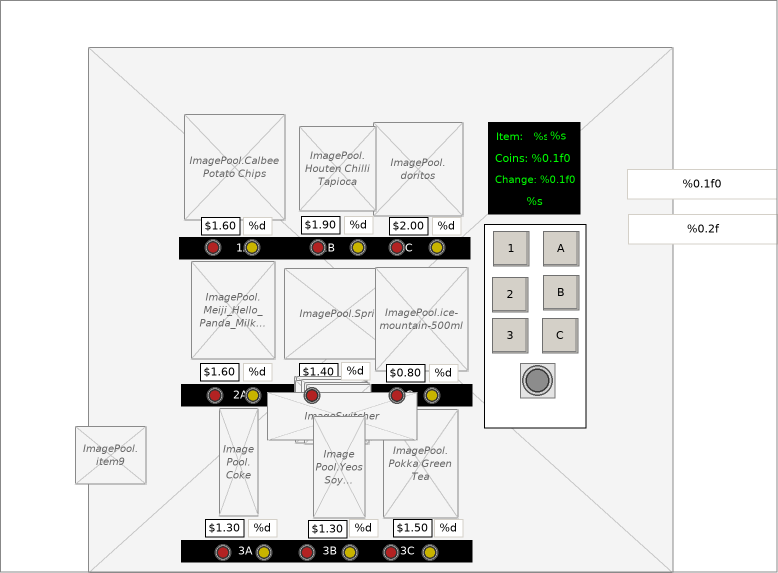
VISUALIZATION Vendingm  // 778x573
    Image (88,47 585x526), image: ImagePool.vending
    Image (184,114 101x106), image: ImagePool.Calbee Potato Chips
    Image (219,408 39x108), image: ImagePool.Coke
    Image (373,122 90x94), image: ImagePool.doritos
    Image (299,126 77x85), image: ImagePool.Houten Chilli Tapioca
    Image (284,268 116x91), image: ImagePool.Sprite
    Image (375,267 93x104), image: ImagePool.ice-mountain-500ml
    Image (383,409 75x109), image: ImagePool.Pokka Green Tea
    Image (191,261 84x98), image: ImagePool.Meiji_Hello_Panda_Milk_Biscuits
    Rectangle (484,224 102x204)
    Button (493,231 36x35), "1"
        tap GVL.button1
    Button (492,277 36x35), "2"
        tap GVL.button2
    Button (543,231 36x35), "A"
        tap GVL.buttonA
    Button (543,275 36x35), "B"
        tap GVL.buttonB
    Button (492,318 36x35), "3"
        tap GVL.button3
    Button (542,318 36x35), "C"
        tap GVL.buttonC
    Rectangle (488,122 92x92)
    Rectangle (179,237 291x22), "1A 1B 1C"
    Rectangle (181,384 291x22), "2A 2B 2C"
    Rectangle (181,540 291x22), "3A 3B 3C"
    Rectangle (201,217 39x18), "$1.60"
    Rectangle (301,216 39x18), "$1.90"
    Rectangle (200,363 39x18), "$1.60"
    Rectangle (308,520 39x18), "$1.30"
    Rectangle (386,364 39x18), "$0.80"
    Rectangle (389,217 39x18), "$2.00"
    Rectangle (299,363 39x18), "$1.40"
    Rectangle (205,519 39x18), "$1.30"
    Rectangle (393,519 39x18), "$1.50"
    Lamp1 (242,238 20x19), variable: GVL.led[1], style: Lamp-Lamp1-Yellow
    Lamp1 (348,238 20x19), variable: GVL.led[2], style: Lamp-Lamp1-Yellow
    Lamp1 (427,238 20x19), variable: GVL.led[3], style: Lamp-Lamp1-Yellow
    Lamp1 (243,386 20x19), variable: GVL.led[4], style: Lamp-Lamp1-Yellow
    Lamp1 (340,386 20x19), variable: GVL.led[5], style: Lamp-Lamp1-Yellow
    Lamp1 (422,386 20x19), variable: GVL.led[6], style: Lamp-Lamp1-Yellow
    Lamp1 (254,543 20x19), variable: GVL.led[7], style: Lamp-Lamp1-Yellow
    Lamp1 (340,543 20x19), variable: GVL.led[8], style: Lamp-Lamp1-Yellow
    Lamp1 (420,543 20x19), variable: GVL.led[9], style: Lamp-Lamp1-Yellow
    Rectangle (493,125 55x23), "Item: %s", text variable: GVL.number
    Rectangle (547,126 29x20), "%s", text variable: GVL.letter
    Rectangle (492,191 85x21), "%s", text variable: GVL.sufficiency
    Image (297,379 70x57), image: ImagePool.item1
        p3560616238: GVL.xvar[1]
        p2738717112: GVL.yvar[1]
    Image (294,376 67x60), image: ImagePool.item2
        p3560616238: GVL.xvar[2]
        p2738717112: GVL.yvar[2]
    Image (296,376 66x58), image: ImagePool.item3
        p3560616238: GVL.xvar[3]
        p2738717112: GVL.yvar[3]
    Image (295,381 65x52), image: ImagePool.item4
        p3560616238: GVL.xvar[4]
        p2738717112: GVL.yvar[4]
    Image (295,380 71x63), image: ImagePool.item5
        p3560616238: GVL.xvar[5]
        p2738717112: GVL.yvar[5]
    Image (301,379 64x58), image: ImagePool.item6
        p3560616238: GVL.xvar[6]
        p2738717112: GVL.yvar[6]
    Image (304,382 65x62), image: ImagePool.item7
        p3560616238: GVL.xvar[7]
        p2738717112: GVL.yvar[7]
    Image (306,384 65x56), image: ImagePool.item8
        p3560616238: GVL.xvar[8]
        p2738717112: GVL.xvar[8]
    Image (75,426 71x58), image: ImagePool.item9
        p3560616238: GVL.xvar[9]
        p2738717112: GVL.yvar[9]
    ImageSwitcher (267,392 150x48), variable: GVL.take, behaviour: TAP
    Rectangle (492,147 85x23), "Coins: %0.1f0", text variable: GVL.dcoins
    Rectangle (492,169 85x21), "Change: %0.1f0", text variable: GVL.dchange
    PushSwitch (520,362 35x37), variable: GVL.buttonO, behaviour: TOGGLE, style: Switch-PushSwitch-Gray
    Textfield (627,169 150x30), "%0.1f0", text variable: MAIN.vending.fbVending1.coinsinsert
        OnMouseClick: write the text variable via Default
    Image (313,416 52x102), image: ImagePool.Yeos Soya Bean Milk
    Textfield (344,216 29x18), "%d", text variable: MAIN.vending.fbVending1.stock[1]
        OnMouseClick: write the text variable via Default
    Textfield (243,217 29x18), "%d", text variable: MAIN.vending.fbVending1.stock[0]
        OnMouseClick: write the text variable via Default
    Textfield (432,217 29x18), "%d", text variable: MAIN.vending.fbVending1.stock[2]
        OnMouseClick: write the text variable via Default
    Textfield (243,363 29x18), "%d", text variable: MAIN.vending.fbVending1.stock[3]
        OnMouseClick: write the text variable via Default
    Textfield (341,362 29x18), "%d", text variable: MAIN.vending.fbVending1.stock[4]
        OnMouseClick: write the text variable via Default
    Textfield (429,364 29x18), "%d", text variable: MAIN.vending.fbVending1.stock[5]
        OnMouseClick: write the text variable via Default
    Textfield (349,519 29x18), "%d", text variable: MAIN.vending.fbVending1.stock[7]
        OnMouseClick: write the text variable via Default
    Textfield (248,519 29x18), "%d", text variable: MAIN.vending.fbVending1.stock[6]
        OnMouseClick: write the text variable via Default
    Textfield (434,519 29x18), "%d", text variable: MAIN.vending.fbVending1.stock[8]
        OnMouseClick: write the text variable via Default
    Textfield (628,214 150x30), "%0.2f", text variable: MAIN.vending.fbVending1.Logistic.sales
        OnMouseClick: write the text variable via Default
    Lamp1 (203,238 20x19), variable: GVL.osled[0], style: Lamp-Lamp1-Red
    Lamp1 (308,238 20x19), variable: GVL.osled[1], style: Lamp-Lamp1-Red
    Lamp1 (205,386 20x19), variable: GVL.osled[3], style: Lamp-Lamp1-Red
    Lamp1 (302,386 20x19), variable: GVL.osled[4], style: Lamp-Lamp1-Red
    Lamp1 (387,386 20x19), variable: GVL.osled[5], style: Lamp-Lamp1-Red
    Lamp1 (213,543 20x19), variable: GVL.osled[6], style: Lamp-Lamp1-Red
    Lamp1 (297,543 20x19), variable: GVL.osled[7], style: Lamp-Lamp1-Red
    Lamp1 (381,543 20x19), variable: GVL.osled[8], style: Lamp-Lamp1-Red
    Lamp1 (387,238 20x19), variable: GVL.osled[2], style: Lamp-Lamp1-Red
END_VISUALIZATION

(* stored: Version 1.1.0.1, ProductVersion 3.1.4024.10
   Visu Vendingm: Id {2e232823-f2d1-412c-a9ba-37116a09e90e} *)
